// TIA Portal V21 export
FUNCTION "HPHV" : Void   // FC11, LAD
{ S7_Optimized_Access := 'TRUE' }
// stored: SetENOAutomatically false
   VAR_TEMP
      "HOLD START" : Bool;
   END_VAR
   VAR_TEMP   // added for the SCL form of the ladder/FBD networks
      _w1 : Bool;
      _w2 : Bool;
      _w3 : Bool;
      _w4 : Bool;
   END_VAR
BEGIN

REGION Network 1
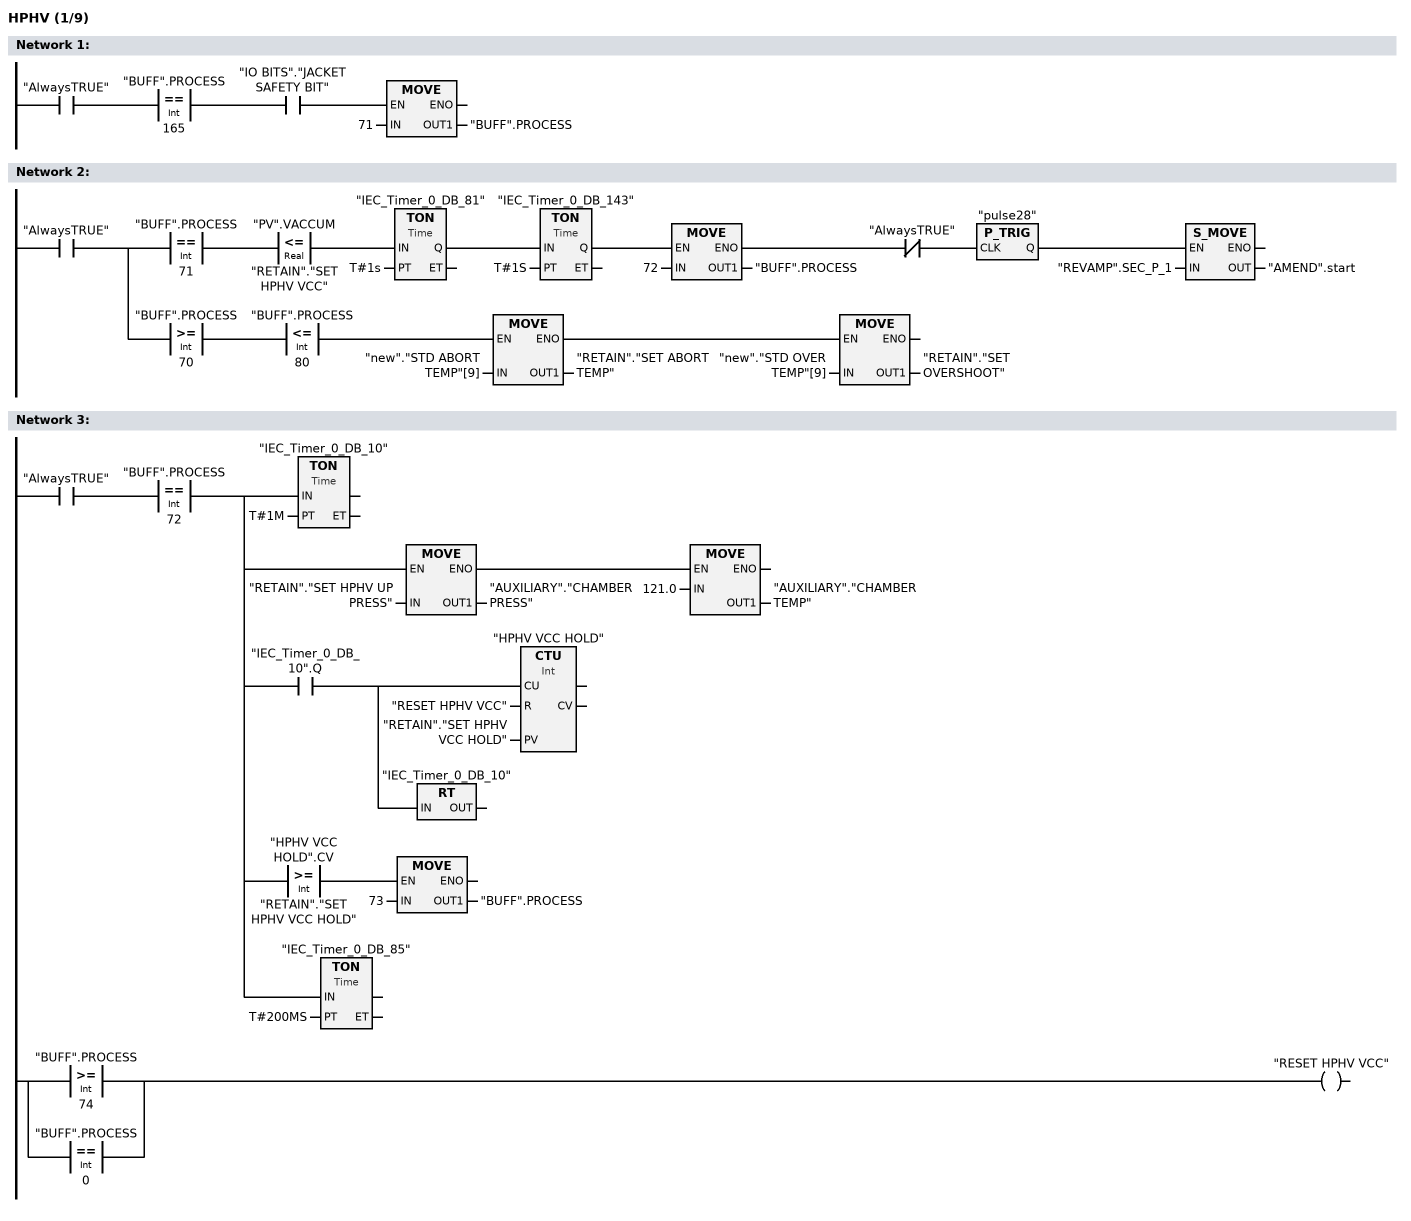
   RUNG wire#powerrail
      Contact( "AlwaysTRUE" )
      { S7_Templates := "SrcType := Int" } EQ_Contact(in1 := "BUFF".PROCESS, in2 := 165)
      Contact( "IO BITS"."JACKET SAFETY BIT" )
      Move(in := 71, out1 => "BUFF".PROCESS)
   END_RUNG
   // the same network as SCL:
   IF "AlwaysTRUE" AND ("BUFF".PROCESS = 165) AND "IO BITS"."JACKET SAFETY BIT" THEN
       "BUFF".PROCESS := 71;
   END_IF;
END_REGION

REGION Network 2
   RUNG wire#powerrail
      Contact( "AlwaysTRUE" )
      wire#w1
      { S7_Templates := "SrcType := Int" } EQ_Contact(in1 := "BUFF".PROCESS, in2 := 71)
      { S7_Templates := "SrcType := Real" } LE_Contact(in1 := "PV".VACCUM, in2 := "RETAIN"."SET HPHV VCC")
      { S7_Templates := "time_type := Time" } "IEC_Timer_0_DB_81".TON(pt := T#1s, et =>)
      { S7_Templates := "time_type := Time" } "IEC_Timer_0_DB_143".TON(pt := T#1S, et =>)
      Move(in := 72, out1 => "BUFF".PROCESS)
      I_Contact( "AlwaysTRUE" )
      P_Trig( "pulse28" )
      S_Move(in := "REVAMP".SEC_P_1, out => "AMEND".start)
   END_RUNG
   RUNG wire#w1
      { S7_Templates := "SrcType := Int" } GE_Contact(in1 := "BUFF".PROCESS, in2 := 70)
      { S7_Templates := "SrcType := Int" } LE_Contact(in1 := "BUFF".PROCESS, in2 := 80)
      Move(in := "new"."STD ABORT TEMP"[9], out1 => "RETAIN"."SET ABORT TEMP")
      Move(in := "new"."STD OVER TEMP"[9], out1 => "RETAIN"."SET OVERSHOOT")
   END_RUNG
   // the same network as SCL:
   "IEC_Timer_0_DB_81".TON(IN := "AlwaysTRUE" AND ("BUFF".PROCESS = 71) AND ("PV".VACCUM <= "RETAIN"."SET HPHV VCC"),
                           PT := T#1s);
   "IEC_Timer_0_DB_143".TON(IN := "IEC_Timer_0_DB_81".Q, PT := T#1S);
   IF "IEC_Timer_0_DB_143".Q THEN "BUFF".PROCESS := 72; END_IF;
   #_w1 := "IEC_Timer_0_DB_143".Q AND NOT "AlwaysTRUE";
   #_w2 := #_w1 AND NOT "pulse28";   // rising edge
   "pulse28" := #_w1;
   IF #_w2 THEN "AMEND".start := "REVAMP".SEC_P_1; END_IF;
   IF "AlwaysTRUE" AND ("BUFF".PROCESS >= 70) AND ("BUFF".PROCESS <= 80) THEN
       "RETAIN"."SET ABORT TEMP" := "new"."STD ABORT TEMP"[9];
       "RETAIN"."SET OVERSHOOT" := "new"."STD OVER TEMP"[9];
   END_IF;
END_REGION

REGION Network 3
   RUNG wire#powerrail
      Contact( "AlwaysTRUE" )
      { S7_Templates := "SrcType := Int" } EQ_Contact(in1 := "BUFF".PROCESS, in2 := 72)
      wire#w1
      { S7_Templates := "time_type := Time" } "IEC_Timer_0_DB_10".TON(pt := T#1M, et =>)
   END_RUNG
   RUNG wire#w1
      Move(in := "RETAIN"."SET HPHV UP PRESS", out1 => "AUXILIARY"."CHAMBER PRESS")
      Move(in := 121.0, out1 => "AUXILIARY"."CHAMBER TEMP")
   END_RUNG
   RUNG wire#w1
      Contact( "IEC_Timer_0_DB_10".Q )
      wire#w2
      { S7_Templates := "value_type := Int" } "HPHV VCC HOLD".CTU(r := "RESET HPHV VCC", pv := "RETAIN"."SET HPHV VCC HOLD", cv =>)
   END_RUNG
   RUNG wire#w2
      RT_Coil( "IEC_Timer_0_DB_10" )
   END_RUNG
   RUNG wire#w1
      { S7_Templates := "SrcType := Int" } GE_Contact(in1 := "HPHV VCC HOLD".CV, in2 := "RETAIN"."SET HPHV VCC HOLD")
      Move(in := 73, out1 => "BUFF".PROCESS)
   END_RUNG
   RUNG wire#w1
      { S7_Templates := "time_type := Time" } "IEC_Timer_0_DB_85".TON(pt := T#200MS, et =>)
   END_RUNG
   RUNG wire#powerrail
      { S7_Templates := "SrcType := Int" } GE_Contact(in1 := "BUFF".PROCESS, in2 := 74)
      wire#w3
      Coil( "RESET HPHV VCC" )
   END_RUNG
   RUNG wire#powerrail
      { S7_Templates := "SrcType := Int" } EQ_Contact(in1 := "BUFF".PROCESS, in2 := 0)
   END_RUNG wire#w3
   // the same network as SCL:
   #_w1 := "AlwaysTRUE" AND ("BUFF".PROCESS = 72);
   "IEC_Timer_0_DB_10".TON(IN := #_w1, PT := T#1M);
   IF #_w1 THEN
       "AUXILIARY"."CHAMBER PRESS" := "RETAIN"."SET HPHV UP PRESS";
       "AUXILIARY"."CHAMBER TEMP" := 121.0;
   END_IF;
   #_w2 := #_w1 AND "IEC_Timer_0_DB_10".Q;
   "HPHV VCC HOLD".CTU(CU := #_w2, R := "RESET HPHV VCC", PV := "RETAIN"."SET HPHV VCC HOLD");
   IF #_w2 THEN RESET_TIMER("IEC_Timer_0_DB_10"); END_IF;
   IF #_w1 AND ("HPHV VCC HOLD".CV >= "RETAIN"."SET HPHV VCC HOLD") THEN "BUFF".PROCESS := 73; END_IF;
   "IEC_Timer_0_DB_85".TON(IN := #_w1, PT := T#200MS);
   "RESET HPHV VCC" := ("BUFF".PROCESS >= 74) OR ("BUFF".PROCESS = 0);
END_REGION

REGION Network 4
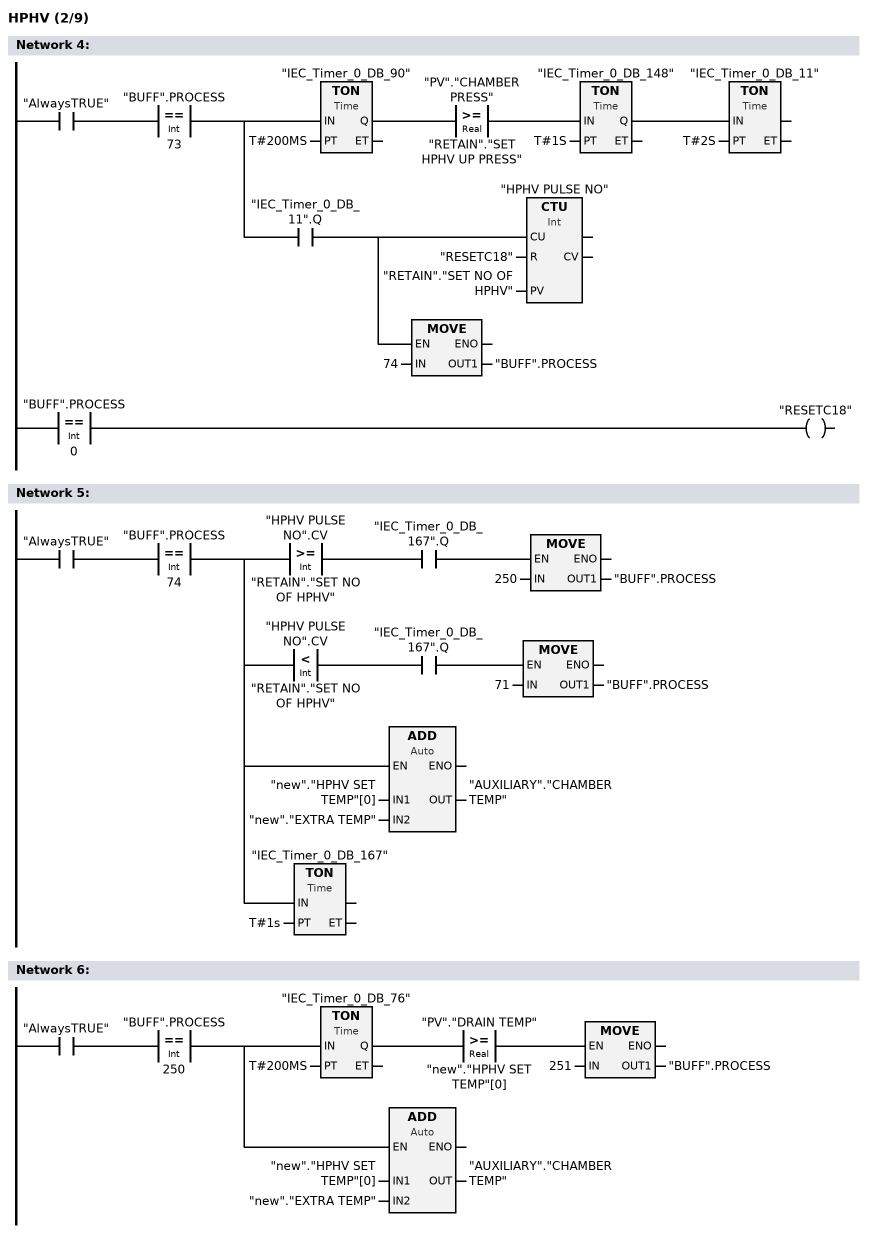
   RUNG wire#powerrail
      Contact( "AlwaysTRUE" )
      { S7_Templates := "SrcType := Int" } EQ_Contact(in1 := "BUFF".PROCESS, in2 := 73)
      wire#w1
      { S7_Templates := "time_type := Time" } "IEC_Timer_0_DB_90".TON(pt := T#200MS, et =>)
      { S7_Templates := "SrcType := Real" } GE_Contact(in1 := "PV"."CHAMBER PRESS", in2 := "RETAIN"."SET HPHV UP PRESS")
      { S7_Templates := "time_type := Time" } "IEC_Timer_0_DB_148".TON(pt := T#1S, et =>)
      { S7_Templates := "time_type := Time" } "IEC_Timer_0_DB_11".TON(pt := T#2S, et =>)
   END_RUNG
   RUNG wire#w1
      Contact( "IEC_Timer_0_DB_11".Q )
      wire#w2
      { S7_Templates := "value_type := Int" } "HPHV PULSE NO".CTU(r := "RESETC18", pv := "RETAIN"."SET NO OF HPHV", cv =>)
   END_RUNG
   RUNG wire#w2
      Move(in := 74, out1 => "BUFF".PROCESS)
   END_RUNG
   RUNG wire#powerrail
      { S7_Templates := "SrcType := Int" } EQ_Contact(in1 := "BUFF".PROCESS, in2 := 0)
      Coil( "RESETC18" )
   END_RUNG
   // the same network as SCL:
   #_w1 := "AlwaysTRUE" AND ("BUFF".PROCESS = 73);
   "IEC_Timer_0_DB_90".TON(IN := #_w1, PT := T#200MS);
   "IEC_Timer_0_DB_148".TON(IN := "IEC_Timer_0_DB_90".Q AND ("PV"."CHAMBER PRESS" >= "RETAIN"."SET HPHV UP PRESS"),
                           PT := T#1S);
   "IEC_Timer_0_DB_11".TON(IN := "IEC_Timer_0_DB_148".Q, PT := T#2S);
   #_w2 := #_w1 AND "IEC_Timer_0_DB_11".Q;
   "HPHV PULSE NO".CTU(CU := #_w2, R := "RESETC18", PV := "RETAIN"."SET NO OF HPHV");
   IF #_w2 THEN "BUFF".PROCESS := 74; END_IF;
   "RESETC18" := "BUFF".PROCESS = 0;
END_REGION

REGION Network 5
   RUNG wire#powerrail
      Contact( "AlwaysTRUE" )
      { S7_Templates := "SrcType := Int" } EQ_Contact(in1 := "BUFF".PROCESS, in2 := 74)
      wire#w1
      { S7_Templates := "SrcType := Int" } GE_Contact(in1 := "HPHV PULSE NO".CV, in2 := "RETAIN"."SET NO OF HPHV")
      Contact( "IEC_Timer_0_DB_167".Q )
      Move(in := 250, out1 => "BUFF".PROCESS)
   END_RUNG
   RUNG wire#w1
      { S7_Templates := "SrcType := Int" } LT_Contact(in1 := "HPHV PULSE NO".CV, in2 := "RETAIN"."SET NO OF HPHV")
      Contact( "IEC_Timer_0_DB_167".Q )
      Move(in := 71, out1 => "BUFF".PROCESS)
   END_RUNG
   RUNG wire#w1
      Add(in1 := "new"."HPHV SET TEMP"[0], in2 := "new"."EXTRA TEMP", out => "AUXILIARY"."CHAMBER TEMP")
   END_RUNG
   RUNG wire#w1
      { S7_Templates := "time_type := Time" } "IEC_Timer_0_DB_167".TON(pt := T#1s, et =>)
   END_RUNG
   // the same network as SCL:
   #_w1 := "AlwaysTRUE" AND ("BUFF".PROCESS = 74);
   IF #_w1 AND ("HPHV PULSE NO".CV >= "RETAIN"."SET NO OF HPHV") AND "IEC_Timer_0_DB_167".Q THEN
       "BUFF".PROCESS := 250;
   END_IF;
   IF #_w1 AND ("HPHV PULSE NO".CV < "RETAIN"."SET NO OF HPHV") AND "IEC_Timer_0_DB_167".Q THEN
       "BUFF".PROCESS := 71;
   END_IF;
   IF #_w1 THEN "AUXILIARY"."CHAMBER TEMP" := "new"."HPHV SET TEMP"[0] + "new"."EXTRA TEMP"; END_IF;
   "IEC_Timer_0_DB_167".TON(IN := #_w1, PT := T#1s);
END_REGION

REGION Network 6
   RUNG wire#powerrail
      Contact( "AlwaysTRUE" )
      { S7_Templates := "SrcType := Int" } EQ_Contact(in1 := "BUFF".PROCESS, in2 := 250)
      wire#w1
      { S7_Templates := "time_type := Time" } "IEC_Timer_0_DB_76".TON(pt := T#200MS, et =>)
      { S7_Templates := "SrcType := Real" } GE_Contact(in1 := "PV"."DRAIN TEMP", in2 := "new"."HPHV SET TEMP"[0])
      Move(in := 251, out1 => "BUFF".PROCESS)
   END_RUNG
   RUNG wire#w1
      Add(in1 := "new"."HPHV SET TEMP"[0], in2 := "new"."EXTRA TEMP", out => "AUXILIARY"."CHAMBER TEMP")
   END_RUNG
   // the same network as SCL:
   #_w1 := "AlwaysTRUE" AND ("BUFF".PROCESS = 250);
   "IEC_Timer_0_DB_76".TON(IN := #_w1, PT := T#200MS);
   IF "IEC_Timer_0_DB_76".Q AND ("PV"."DRAIN TEMP" >= "new"."HPHV SET TEMP"[0]) THEN
       "BUFF".PROCESS := 251;
   END_IF;
   IF #_w1 THEN "AUXILIARY"."CHAMBER TEMP" := "new"."HPHV SET TEMP"[0] + "new"."EXTRA TEMP"; END_IF;
END_REGION

REGION Network 7
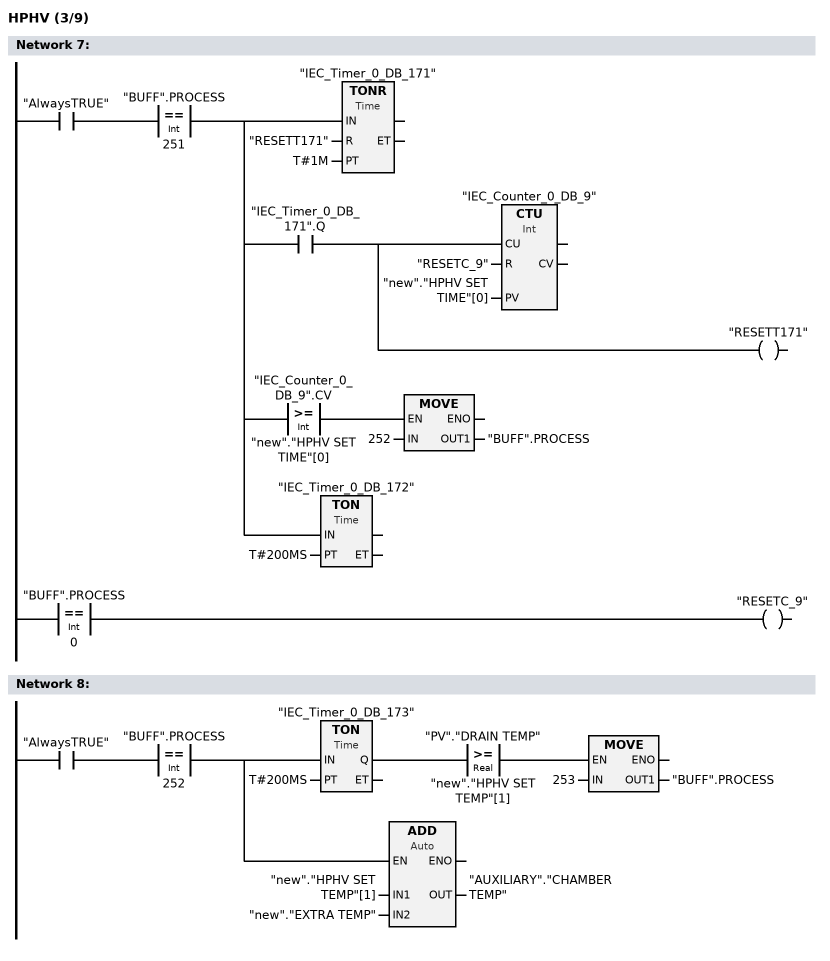
   RUNG wire#powerrail
      Contact( "AlwaysTRUE" )
      { S7_Templates := "SrcType := Int" } EQ_Contact(in1 := "BUFF".PROCESS, in2 := 251)
      wire#w1
      { S7_Templates := "time_type := Time" } "IEC_Timer_0_DB_171".TONR(r := "RESETT171", pt := T#1M, et =>)
   END_RUNG
   RUNG wire#w1
      Contact( "IEC_Timer_0_DB_171".Q )
      wire#w2
      { S7_Templates := "value_type := Int" } "IEC_Counter_0_DB_9".CTU(r := "RESETC_9", pv := "new"."HPHV SET TIME"[0], cv =>)
   END_RUNG
   RUNG wire#w2
      Coil( "RESETT171" )
   END_RUNG
   RUNG wire#w1
      { S7_Templates := "SrcType := Int" } GE_Contact(in1 := "IEC_Counter_0_DB_9".CV, in2 := "new"."HPHV SET TIME"[0])
      Move(in := 252, out1 => "BUFF".PROCESS)
   END_RUNG
   RUNG wire#w1
      { S7_Templates := "time_type := Time" } "IEC_Timer_0_DB_172".TON(pt := T#200MS, et =>)
   END_RUNG
   RUNG wire#powerrail
      { S7_Templates := "SrcType := Int" } EQ_Contact(in1 := "BUFF".PROCESS, in2 := 0)
      Coil( "RESETC_9" )
   END_RUNG
   // the same network as SCL:
   #_w1 := "AlwaysTRUE" AND ("BUFF".PROCESS = 251);
   "IEC_Timer_0_DB_171".TONR(IN := #_w1, R := "RESETT171", PT := T#1M);
   #_w2 := #_w1 AND "IEC_Timer_0_DB_171".Q;
   "IEC_Counter_0_DB_9".CTU(CU := #_w2, R := "RESETC_9", PV := "new"."HPHV SET TIME"[0]);
   "RESETT171" := #_w2;
   IF #_w1 AND ("IEC_Counter_0_DB_9".CV >= "new"."HPHV SET TIME"[0]) THEN "BUFF".PROCESS := 252; END_IF;
   "IEC_Timer_0_DB_172".TON(IN := #_w1, PT := T#200MS);
   "RESETC_9" := "BUFF".PROCESS = 0;
END_REGION

REGION Network 8
   RUNG wire#powerrail
      Contact( "AlwaysTRUE" )
      { S7_Templates := "SrcType := Int" } EQ_Contact(in1 := "BUFF".PROCESS, in2 := 252)
      wire#w1
      { S7_Templates := "time_type := Time" } "IEC_Timer_0_DB_173".TON(pt := T#200MS, et =>)
      { S7_Templates := "SrcType := Real" } GE_Contact(in1 := "PV"."DRAIN TEMP", in2 := "new"."HPHV SET TEMP"[1])
      Move(in := 253, out1 => "BUFF".PROCESS)
   END_RUNG
   RUNG wire#w1
      Add(in1 := "new"."HPHV SET TEMP"[1], in2 := "new"."EXTRA TEMP", out => "AUXILIARY"."CHAMBER TEMP")
   END_RUNG
   // the same network as SCL:
   #_w1 := "AlwaysTRUE" AND ("BUFF".PROCESS = 252);
   "IEC_Timer_0_DB_173".TON(IN := #_w1, PT := T#200MS);
   IF "IEC_Timer_0_DB_173".Q AND ("PV"."DRAIN TEMP" >= "new"."HPHV SET TEMP"[1]) THEN
       "BUFF".PROCESS := 253;
   END_IF;
   IF #_w1 THEN "AUXILIARY"."CHAMBER TEMP" := "new"."HPHV SET TEMP"[1] + "new"."EXTRA TEMP"; END_IF;
END_REGION

REGION Network 9
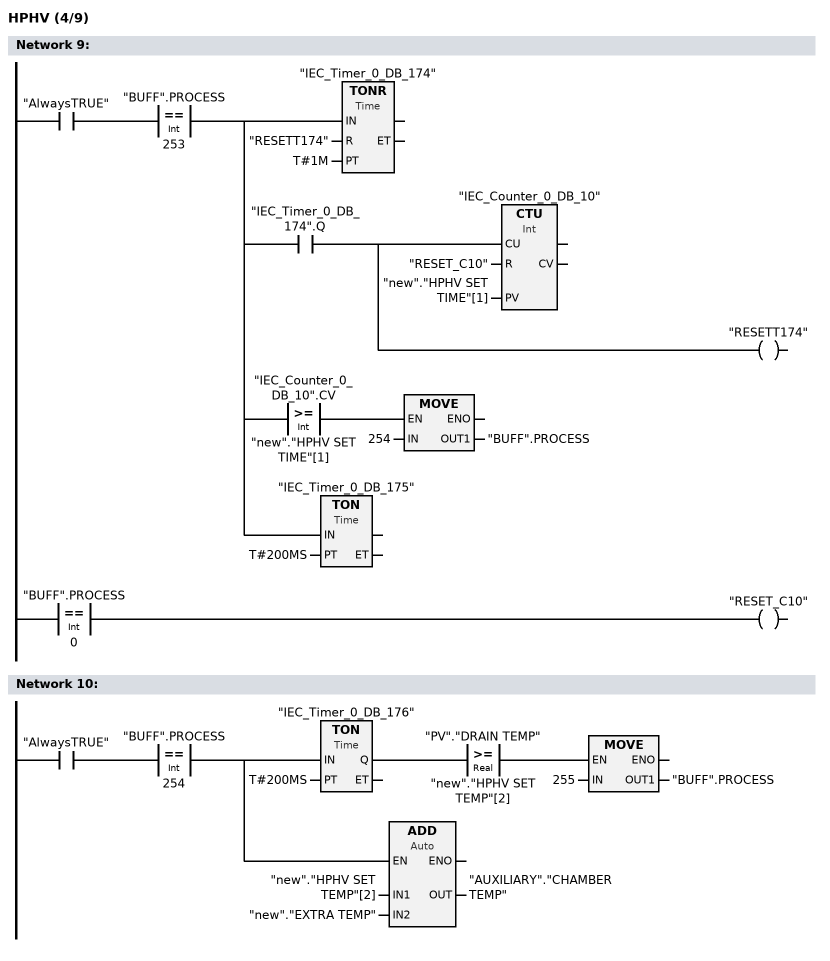
   RUNG wire#powerrail
      Contact( "AlwaysTRUE" )
      { S7_Templates := "SrcType := Int" } EQ_Contact(in1 := "BUFF".PROCESS, in2 := 253)
      wire#w1
      { S7_Templates := "time_type := Time" } "IEC_Timer_0_DB_174".TONR(r := "RESETT174", pt := T#1M, et =>)
   END_RUNG
   RUNG wire#w1
      Contact( "IEC_Timer_0_DB_174".Q )
      wire#w2
      { S7_Templates := "value_type := Int" } "IEC_Counter_0_DB_10".CTU(r := "RESET_C10", pv := "new"."HPHV SET TIME"[1], cv =>)
   END_RUNG
   RUNG wire#w2
      Coil( "RESETT174" )
   END_RUNG
   RUNG wire#w1
      { S7_Templates := "SrcType := Int" } GE_Contact(in1 := "IEC_Counter_0_DB_10".CV, in2 := "new"."HPHV SET TIME"[1])
      Move(in := 254, out1 => "BUFF".PROCESS)
   END_RUNG
   RUNG wire#w1
      { S7_Templates := "time_type := Time" } "IEC_Timer_0_DB_175".TON(pt := T#200MS, et =>)
   END_RUNG
   RUNG wire#powerrail
      { S7_Templates := "SrcType := Int" } EQ_Contact(in1 := "BUFF".PROCESS, in2 := 0)
      Coil( "RESET_C10" )
   END_RUNG
   // the same network as SCL:
   #_w1 := "AlwaysTRUE" AND ("BUFF".PROCESS = 253);
   "IEC_Timer_0_DB_174".TONR(IN := #_w1, R := "RESETT174", PT := T#1M);
   #_w2 := #_w1 AND "IEC_Timer_0_DB_174".Q;
   "IEC_Counter_0_DB_10".CTU(CU := #_w2, R := "RESET_C10", PV := "new"."HPHV SET TIME"[1]);
   "RESETT174" := #_w2;
   IF #_w1 AND ("IEC_Counter_0_DB_10".CV >= "new"."HPHV SET TIME"[1]) THEN "BUFF".PROCESS := 254; END_IF;
   "IEC_Timer_0_DB_175".TON(IN := #_w1, PT := T#200MS);
   "RESET_C10" := "BUFF".PROCESS = 0;
END_REGION

REGION Network 10
   RUNG wire#powerrail
      Contact( "AlwaysTRUE" )
      { S7_Templates := "SrcType := Int" } EQ_Contact(in1 := "BUFF".PROCESS, in2 := 254)
      wire#w1
      { S7_Templates := "time_type := Time" } "IEC_Timer_0_DB_176".TON(pt := T#200MS, et =>)
      { S7_Templates := "SrcType := Real" } GE_Contact(in1 := "PV"."DRAIN TEMP", in2 := "new"."HPHV SET TEMP"[2])
      Move(in := 255, out1 => "BUFF".PROCESS)
   END_RUNG
   RUNG wire#w1
      Add(in1 := "new"."HPHV SET TEMP"[2], in2 := "new"."EXTRA TEMP", out => "AUXILIARY"."CHAMBER TEMP")
   END_RUNG
   // the same network as SCL:
   #_w1 := "AlwaysTRUE" AND ("BUFF".PROCESS = 254);
   "IEC_Timer_0_DB_176".TON(IN := #_w1, PT := T#200MS);
   IF "IEC_Timer_0_DB_176".Q AND ("PV"."DRAIN TEMP" >= "new"."HPHV SET TEMP"[2]) THEN
       "BUFF".PROCESS := 255;
   END_IF;
   IF #_w1 THEN "AUXILIARY"."CHAMBER TEMP" := "new"."HPHV SET TEMP"[2] + "new"."EXTRA TEMP"; END_IF;
END_REGION

REGION Network 11
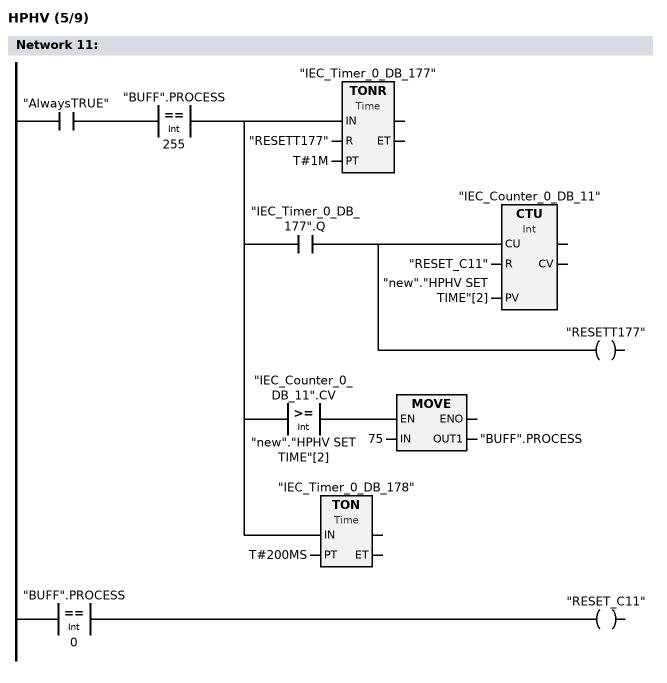
   RUNG wire#powerrail
      Contact( "AlwaysTRUE" )
      { S7_Templates := "SrcType := Int" } EQ_Contact(in1 := "BUFF".PROCESS, in2 := 255)
      wire#w1
      { S7_Templates := "time_type := Time" } "IEC_Timer_0_DB_177".TONR(r := "RESETT177", pt := T#1M, et =>)
   END_RUNG
   RUNG wire#w1
      Contact( "IEC_Timer_0_DB_177".Q )
      wire#w2
      { S7_Templates := "value_type := Int" } "IEC_Counter_0_DB_11".CTU(r := "RESET_C11", pv := "new"."HPHV SET TIME"[2], cv =>)
   END_RUNG
   RUNG wire#w2
      Coil( "RESETT177" )
   END_RUNG
   RUNG wire#w1
      { S7_Templates := "SrcType := Int" } GE_Contact(in1 := "IEC_Counter_0_DB_11".CV, in2 := "new"."HPHV SET TIME"[2])
      Move(in := 75, out1 => "BUFF".PROCESS)
   END_RUNG
   RUNG wire#w1
      { S7_Templates := "time_type := Time" } "IEC_Timer_0_DB_178".TON(pt := T#200MS, et =>)
   END_RUNG
   RUNG wire#powerrail
      { S7_Templates := "SrcType := Int" } EQ_Contact(in1 := "BUFF".PROCESS, in2 := 0)
      Coil( "RESET_C11" )
   END_RUNG
   // the same network as SCL:
   #_w1 := "AlwaysTRUE" AND ("BUFF".PROCESS = 255);
   "IEC_Timer_0_DB_177".TONR(IN := #_w1, R := "RESETT177", PT := T#1M);
   #_w2 := #_w1 AND "IEC_Timer_0_DB_177".Q;
   "IEC_Counter_0_DB_11".CTU(CU := #_w2, R := "RESET_C11", PV := "new"."HPHV SET TIME"[2]);
   "RESETT177" := #_w2;
   IF #_w1 AND ("IEC_Counter_0_DB_11".CV >= "new"."HPHV SET TIME"[2]) THEN "BUFF".PROCESS := 75; END_IF;
   "IEC_Timer_0_DB_178".TON(IN := #_w1, PT := T#200MS);
   "RESET_C11" := "BUFF".PROCESS = 0;
END_REGION

REGION Network 12
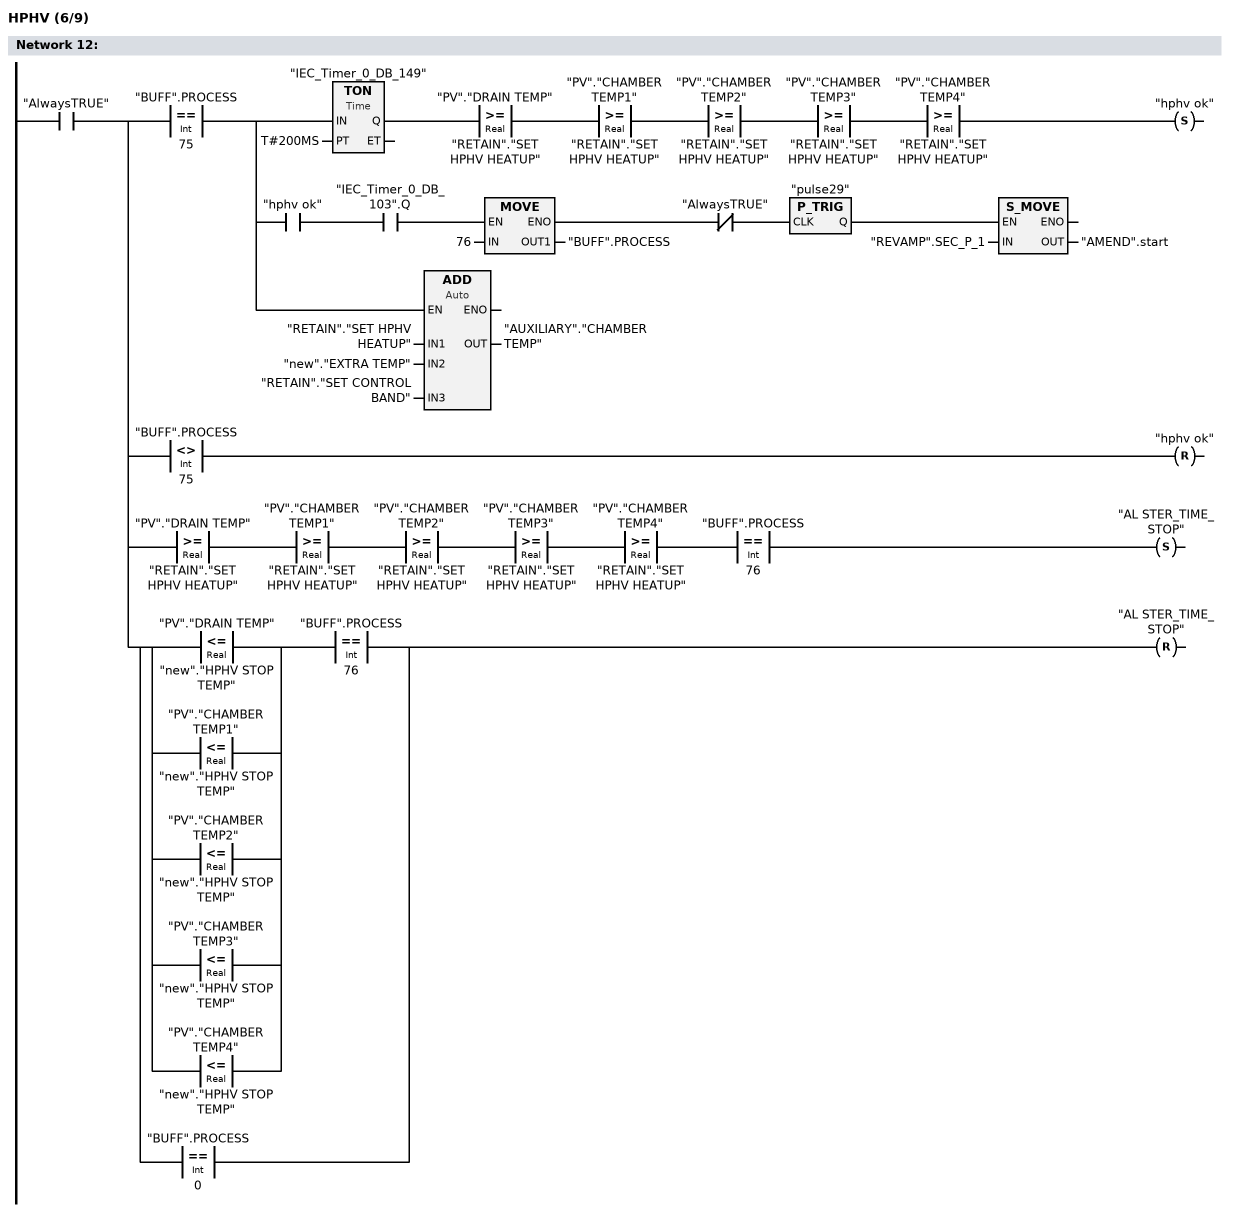
   RUNG wire#powerrail
      Contact( "AlwaysTRUE" )
      wire#w1
      { S7_Templates := "SrcType := Int" } EQ_Contact(in1 := "BUFF".PROCESS, in2 := 75)
      wire#w2
      { S7_Templates := "time_type := Time" } "IEC_Timer_0_DB_149".TON(pt := T#200MS, et =>)
      { S7_Templates := "SrcType := Real" } GE_Contact(in1 := "PV"."DRAIN TEMP", in2 := "RETAIN"."SET HPHV HEATUP")
      { S7_Templates := "SrcType := Real" } GE_Contact(in1 := "PV"."CHAMBER TEMP1", in2 := "RETAIN"."SET HPHV HEATUP")
      { S7_Templates := "SrcType := Real" } GE_Contact(in1 := "PV"."CHAMBER TEMP2", in2 := "RETAIN"."SET HPHV HEATUP")
      { S7_Templates := "SrcType := Real" } GE_Contact(in1 := "PV"."CHAMBER TEMP3", in2 := "RETAIN"."SET HPHV HEATUP")
      { S7_Templates := "SrcType := Real" } GE_Contact(in1 := "PV"."CHAMBER TEMP4", in2 := "RETAIN"."SET HPHV HEATUP")
      S_Coil( "hphv ok" )
   END_RUNG
   RUNG wire#w2
      Contact( "hphv ok" )
      Contact( "IEC_Timer_0_DB_103".Q )
      Move(in := 76, out1 => "BUFF".PROCESS)
      I_Contact( "AlwaysTRUE" )
      P_Trig( "pulse29" )
      S_Move(in := "REVAMP".SEC_P_1, out => "AMEND".start)
   END_RUNG
   RUNG wire#w2
      Add(in1 := "RETAIN"."SET HPHV HEATUP", in2 := "new"."EXTRA TEMP", in3 := "RETAIN"."SET CONTROL BAND", out => "AUXILIARY"."CHAMBER TEMP")
   END_RUNG
   RUNG wire#w1
      { S7_Templates := "SrcType := Int" } NE_Contact(in1 := "BUFF".PROCESS, in2 := 75)
      R_Coil( "hphv ok" )
   END_RUNG
   RUNG wire#w1
      { S7_Templates := "SrcType := Real" } GE_Contact(in1 := "PV"."DRAIN TEMP", in2 := "RETAIN"."SET HPHV HEATUP")
      { S7_Templates := "SrcType := Real" } GE_Contact(in1 := "PV"."CHAMBER TEMP1", in2 := "RETAIN"."SET HPHV HEATUP")
      { S7_Templates := "SrcType := Real" } GE_Contact(in1 := "PV"."CHAMBER TEMP2", in2 := "RETAIN"."SET HPHV HEATUP")
      { S7_Templates := "SrcType := Real" } GE_Contact(in1 := "PV"."CHAMBER TEMP3", in2 := "RETAIN"."SET HPHV HEATUP")
      { S7_Templates := "SrcType := Real" } GE_Contact(in1 := "PV"."CHAMBER TEMP4", in2 := "RETAIN"."SET HPHV HEATUP")
      { S7_Templates := "SrcType := Int" } EQ_Contact(in1 := "BUFF".PROCESS, in2 := 76)
      S_Coil( "AL STER_TIME_STOP" )
   END_RUNG
   RUNG wire#w1
      { S7_Templates := "SrcType := Real" } LE_Contact(in1 := "PV"."DRAIN TEMP", in2 := "new"."HPHV STOP TEMP")
      wire#w3
      { S7_Templates := "SrcType := Int" } EQ_Contact(in1 := "BUFF".PROCESS, in2 := 76)
      wire#w4
      R_Coil( "AL STER_TIME_STOP" )
   END_RUNG
   RUNG wire#w1
      { S7_Templates := "SrcType := Real" } LE_Contact(in1 := "PV"."CHAMBER TEMP1", in2 := "new"."HPHV STOP TEMP")
   END_RUNG wire#w3
   RUNG wire#w1
      { S7_Templates := "SrcType := Real" } LE_Contact(in1 := "PV"."CHAMBER TEMP2", in2 := "new"."HPHV STOP TEMP")
   END_RUNG wire#w3
   RUNG wire#w1
      { S7_Templates := "SrcType := Real" } LE_Contact(in1 := "PV"."CHAMBER TEMP3", in2 := "new"."HPHV STOP TEMP")
   END_RUNG wire#w3
   RUNG wire#w1
      { S7_Templates := "SrcType := Real" } LE_Contact(in1 := "PV"."CHAMBER TEMP4", in2 := "new"."HPHV STOP TEMP")
   END_RUNG wire#w3
   RUNG wire#w1
      { S7_Templates := "SrcType := Int" } EQ_Contact(in1 := "BUFF".PROCESS, in2 := 0)
   END_RUNG wire#w4
   // the same network as SCL:
   #_w1 := "AlwaysTRUE" AND ("BUFF".PROCESS = 75);
   "IEC_Timer_0_DB_149".TON(IN := #_w1, PT := T#200MS);
   IF "IEC_Timer_0_DB_149".Q AND ("PV"."DRAIN TEMP" >= "RETAIN"."SET HPHV HEATUP") AND ("PV"."CHAMBER TEMP1" >= "RETAIN"."SET HPHV HEATUP") AND ("PV"."CHAMBER TEMP2" >= "RETAIN"."SET HPHV HEATUP") AND ("PV"."CHAMBER TEMP3" >= "RETAIN"."SET HPHV HEATUP") AND ("PV"."CHAMBER TEMP4" >= "RETAIN"."SET HPHV HEATUP") THEN
       "hphv ok" := TRUE;
   END_IF;
   #_w2 := #_w1 AND "hphv ok" AND "IEC_Timer_0_DB_103".Q;
   IF #_w2 THEN "BUFF".PROCESS := 76; END_IF;
   #_w3 := #_w2 AND NOT "AlwaysTRUE";
   #_w4 := #_w3 AND NOT "pulse29";   // rising edge
   "pulse29" := #_w3;
   IF #_w4 THEN "AMEND".start := "REVAMP".SEC_P_1; END_IF;
   IF #_w1 THEN
       "AUXILIARY"."CHAMBER TEMP" := "RETAIN"."SET HPHV HEATUP" + "new"."EXTRA TEMP" + "RETAIN"."SET CONTROL BAND";
   END_IF;
   IF "AlwaysTRUE" AND ("BUFF".PROCESS <> 75) THEN "hphv ok" := FALSE; END_IF;
   IF "AlwaysTRUE" AND ("PV"."DRAIN TEMP" >= "RETAIN"."SET HPHV HEATUP") AND ("PV"."CHAMBER TEMP1" >= "RETAIN"."SET HPHV HEATUP") AND ("PV"."CHAMBER TEMP2" >= "RETAIN"."SET HPHV HEATUP") AND ("PV"."CHAMBER TEMP3" >= "RETAIN"."SET HPHV HEATUP") AND ("PV"."CHAMBER TEMP4" >= "RETAIN"."SET HPHV HEATUP") AND ("BUFF".PROCESS = 76) THEN
       "AL STER_TIME_STOP" := TRUE;
   END_IF;
   IF "AlwaysTRUE" AND (((("PV"."DRAIN TEMP" <= "new"."HPHV STOP TEMP") OR ("PV"."CHAMBER TEMP1" <= "new"."HPHV STOP TEMP") OR ("PV"."CHAMBER TEMP2" <= "new"."HPHV STOP TEMP") OR ("PV"."CHAMBER TEMP3" <= "new"."HPHV STOP TEMP") OR ("PV"."CHAMBER TEMP4" <= "new"."HPHV STOP TEMP")) AND ("BUFF".PROCESS = 76)) OR ("BUFF".PROCESS = 0)) THEN
       "AL STER_TIME_STOP" := FALSE;
   END_IF;
END_REGION

REGION Network 13
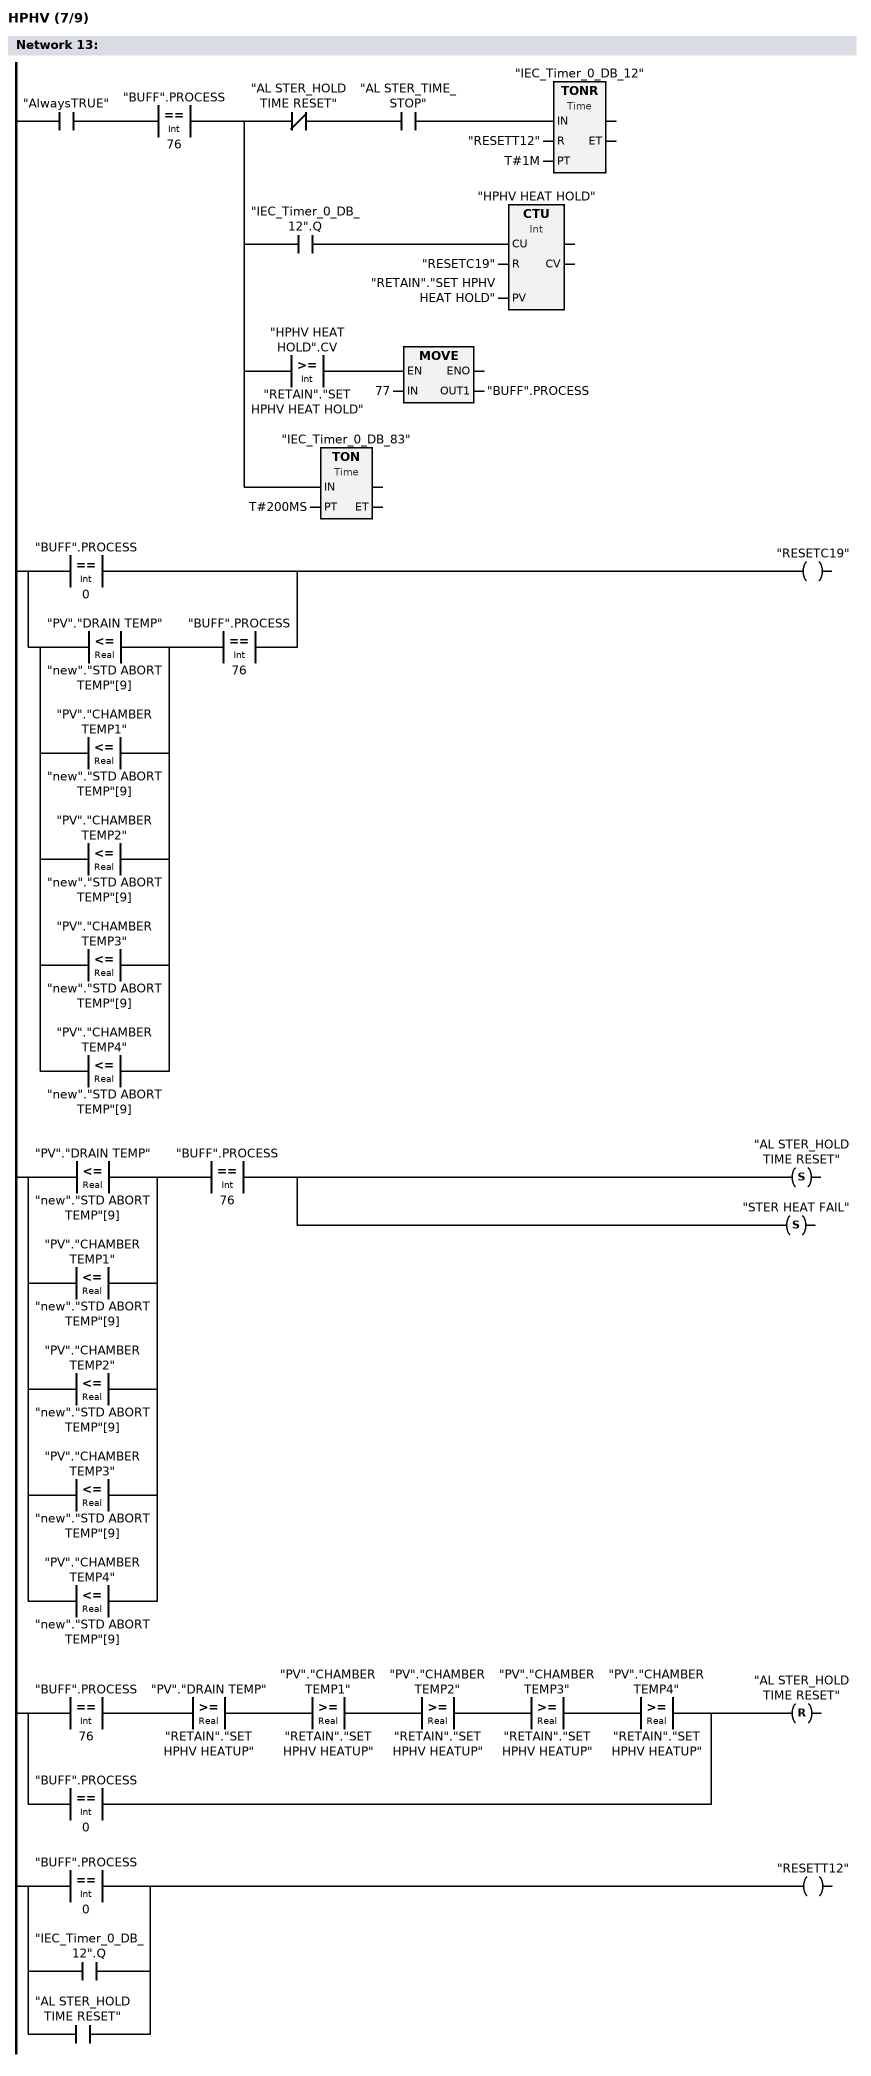
   RUNG wire#powerrail
      Contact( "AlwaysTRUE" )
      { S7_Templates := "SrcType := Int" } EQ_Contact(in1 := "BUFF".PROCESS, in2 := 76)
      wire#w1
      I_Contact( "AL STER_HOLD TIME RESET" )
      Contact( "AL STER_TIME_STOP" )
      { S7_Templates := "time_type := Time" } "IEC_Timer_0_DB_12".TONR(r := "RESETT12", pt := T#1M, et =>)
   END_RUNG
   RUNG wire#w1
      Contact( "IEC_Timer_0_DB_12".Q )
      { S7_Templates := "value_type := Int" } "HPHV HEAT HOLD".CTU(r := "RESETC19", pv := "RETAIN"."SET HPHV HEAT HOLD", cv =>)
   END_RUNG
   RUNG wire#w1
      { S7_Templates := "SrcType := Int" } GE_Contact(in1 := "HPHV HEAT HOLD".CV, in2 := "RETAIN"."SET HPHV HEAT HOLD")
      Move(in := 77, out1 => "BUFF".PROCESS)
   END_RUNG
   RUNG wire#w1
      { S7_Templates := "time_type := Time" } "IEC_Timer_0_DB_83".TON(pt := T#200MS, et =>)
   END_RUNG
   RUNG wire#powerrail
      { S7_Templates := "SrcType := Int" } EQ_Contact(in1 := "BUFF".PROCESS, in2 := 0)
      wire#w2
      Coil( "RESETC19" )
   END_RUNG
   RUNG wire#powerrail
      { S7_Templates := "SrcType := Real" } LE_Contact(in1 := "PV"."DRAIN TEMP", in2 := "new"."STD ABORT TEMP"[9])
      wire#w3
      { S7_Templates := "SrcType := Int" } EQ_Contact(in1 := "BUFF".PROCESS, in2 := 76)
   END_RUNG wire#w2
   RUNG wire#powerrail
      { S7_Templates := "SrcType := Real" } LE_Contact(in1 := "PV"."CHAMBER TEMP1", in2 := "new"."STD ABORT TEMP"[9])
   END_RUNG wire#w3
   RUNG wire#powerrail
      { S7_Templates := "SrcType := Real" } LE_Contact(in1 := "PV"."CHAMBER TEMP2", in2 := "new"."STD ABORT TEMP"[9])
   END_RUNG wire#w3
   RUNG wire#powerrail
      { S7_Templates := "SrcType := Real" } LE_Contact(in1 := "PV"."CHAMBER TEMP3", in2 := "new"."STD ABORT TEMP"[9])
   END_RUNG wire#w3
   RUNG wire#powerrail
      { S7_Templates := "SrcType := Real" } LE_Contact(in1 := "PV"."CHAMBER TEMP4", in2 := "new"."STD ABORT TEMP"[9])
   END_RUNG wire#w3
   RUNG wire#powerrail
      { S7_Templates := "SrcType := Real" } LE_Contact(in1 := "PV"."DRAIN TEMP", in2 := "new"."STD ABORT TEMP"[9])
      wire#w4
      { S7_Templates := "SrcType := Int" } EQ_Contact(in1 := "BUFF".PROCESS, in2 := 76)
      wire#w5
      S_Coil( "AL STER_HOLD TIME RESET" )
   END_RUNG
   RUNG wire#powerrail
      { S7_Templates := "SrcType := Real" } LE_Contact(in1 := "PV"."CHAMBER TEMP1", in2 := "new"."STD ABORT TEMP"[9])
   END_RUNG wire#w4
   RUNG wire#powerrail
      { S7_Templates := "SrcType := Real" } LE_Contact(in1 := "PV"."CHAMBER TEMP2", in2 := "new"."STD ABORT TEMP"[9])
   END_RUNG wire#w4
   RUNG wire#powerrail
      { S7_Templates := "SrcType := Real" } LE_Contact(in1 := "PV"."CHAMBER TEMP3", in2 := "new"."STD ABORT TEMP"[9])
   END_RUNG wire#w4
   RUNG wire#powerrail
      { S7_Templates := "SrcType := Real" } LE_Contact(in1 := "PV"."CHAMBER TEMP4", in2 := "new"."STD ABORT TEMP"[9])
   END_RUNG wire#w4
   RUNG wire#w5
      S_Coil( "STER HEAT FAIL" )
   END_RUNG
   RUNG wire#powerrail
      { S7_Templates := "SrcType := Int" } EQ_Contact(in1 := "BUFF".PROCESS, in2 := 76)
      { S7_Templates := "SrcType := Real" } GE_Contact(in1 := "PV"."DRAIN TEMP", in2 := "RETAIN"."SET HPHV HEATUP")
      { S7_Templates := "SrcType := Real" } GE_Contact(in1 := "PV"."CHAMBER TEMP1", in2 := "RETAIN"."SET HPHV HEATUP")
      { S7_Templates := "SrcType := Real" } GE_Contact(in1 := "PV"."CHAMBER TEMP2", in2 := "RETAIN"."SET HPHV HEATUP")
      { S7_Templates := "SrcType := Real" } GE_Contact(in1 := "PV"."CHAMBER TEMP3", in2 := "RETAIN"."SET HPHV HEATUP")
      { S7_Templates := "SrcType := Real" } GE_Contact(in1 := "PV"."CHAMBER TEMP4", in2 := "RETAIN"."SET HPHV HEATUP")
      wire#w6
      R_Coil( "AL STER_HOLD TIME RESET" )
   END_RUNG
   RUNG wire#powerrail
      { S7_Templates := "SrcType := Int" } EQ_Contact(in1 := "BUFF".PROCESS, in2 := 0)
   END_RUNG wire#w6
   RUNG wire#powerrail
      { S7_Templates := "SrcType := Int" } EQ_Contact(in1 := "BUFF".PROCESS, in2 := 0)
      wire#w7
      Coil( "RESETT12" )
   END_RUNG
   RUNG wire#powerrail
      Contact( "IEC_Timer_0_DB_12".Q )
   END_RUNG wire#w7
   RUNG wire#powerrail
      Contact( "AL STER_HOLD TIME RESET" )
   END_RUNG wire#w7
   // the same network as SCL:
   #_w1 := "AlwaysTRUE" AND ("BUFF".PROCESS = 76);
   "IEC_Timer_0_DB_12".TONR(IN := #_w1 AND NOT "AL STER_HOLD TIME RESET" AND "AL STER_TIME_STOP",
                           R := "RESETT12",
                           PT := T#1M);
   "HPHV HEAT HOLD".CTU(CU := #_w1 AND "IEC_Timer_0_DB_12".Q,
                        R := "RESETC19",
                        PV := "RETAIN"."SET HPHV HEAT HOLD");
   IF #_w1 AND ("HPHV HEAT HOLD".CV >= "RETAIN"."SET HPHV HEAT HOLD") THEN "BUFF".PROCESS := 77; END_IF;
   "IEC_Timer_0_DB_83".TON(IN := #_w1, PT := T#200MS);
   "RESETC19" := ("BUFF".PROCESS = 0) OR ((("PV"."DRAIN TEMP" <= "new"."STD ABORT TEMP"[9]) OR ("PV"."CHAMBER TEMP1" <= "new"."STD ABORT TEMP"[9]) OR ("PV"."CHAMBER TEMP2" <= "new"."STD ABORT TEMP"[9]) OR ("PV"."CHAMBER TEMP3" <= "new"."STD ABORT TEMP"[9]) OR ("PV"."CHAMBER TEMP4" <= "new"."STD ABORT TEMP"[9])) AND ("BUFF".PROCESS = 76));
   IF (("PV"."DRAIN TEMP" <= "new"."STD ABORT TEMP"[9]) OR ("PV"."CHAMBER TEMP1" <= "new"."STD ABORT TEMP"[9]) OR ("PV"."CHAMBER TEMP2" <= "new"."STD ABORT TEMP"[9]) OR ("PV"."CHAMBER TEMP3" <= "new"."STD ABORT TEMP"[9]) OR ("PV"."CHAMBER TEMP4" <= "new"."STD ABORT TEMP"[9])) AND ("BUFF".PROCESS = 76) THEN
       "AL STER_HOLD TIME RESET" := TRUE;
       "STER HEAT FAIL" := TRUE;
   END_IF;
   IF (("BUFF".PROCESS = 76) AND ("PV"."DRAIN TEMP" >= "RETAIN"."SET HPHV HEATUP") AND ("PV"."CHAMBER TEMP1" >= "RETAIN"."SET HPHV HEATUP") AND ("PV"."CHAMBER TEMP2" >= "RETAIN"."SET HPHV HEATUP") AND ("PV"."CHAMBER TEMP3" >= "RETAIN"."SET HPHV HEATUP") AND ("PV"."CHAMBER TEMP4" >= "RETAIN"."SET HPHV HEATUP")) OR ("BUFF".PROCESS = 0) THEN
       "AL STER_HOLD TIME RESET" := FALSE;
   END_IF;
   "RESETT12" := ("BUFF".PROCESS = 0) OR "IEC_Timer_0_DB_12".Q OR "AL STER_HOLD TIME RESET";
END_REGION

REGION Network 14
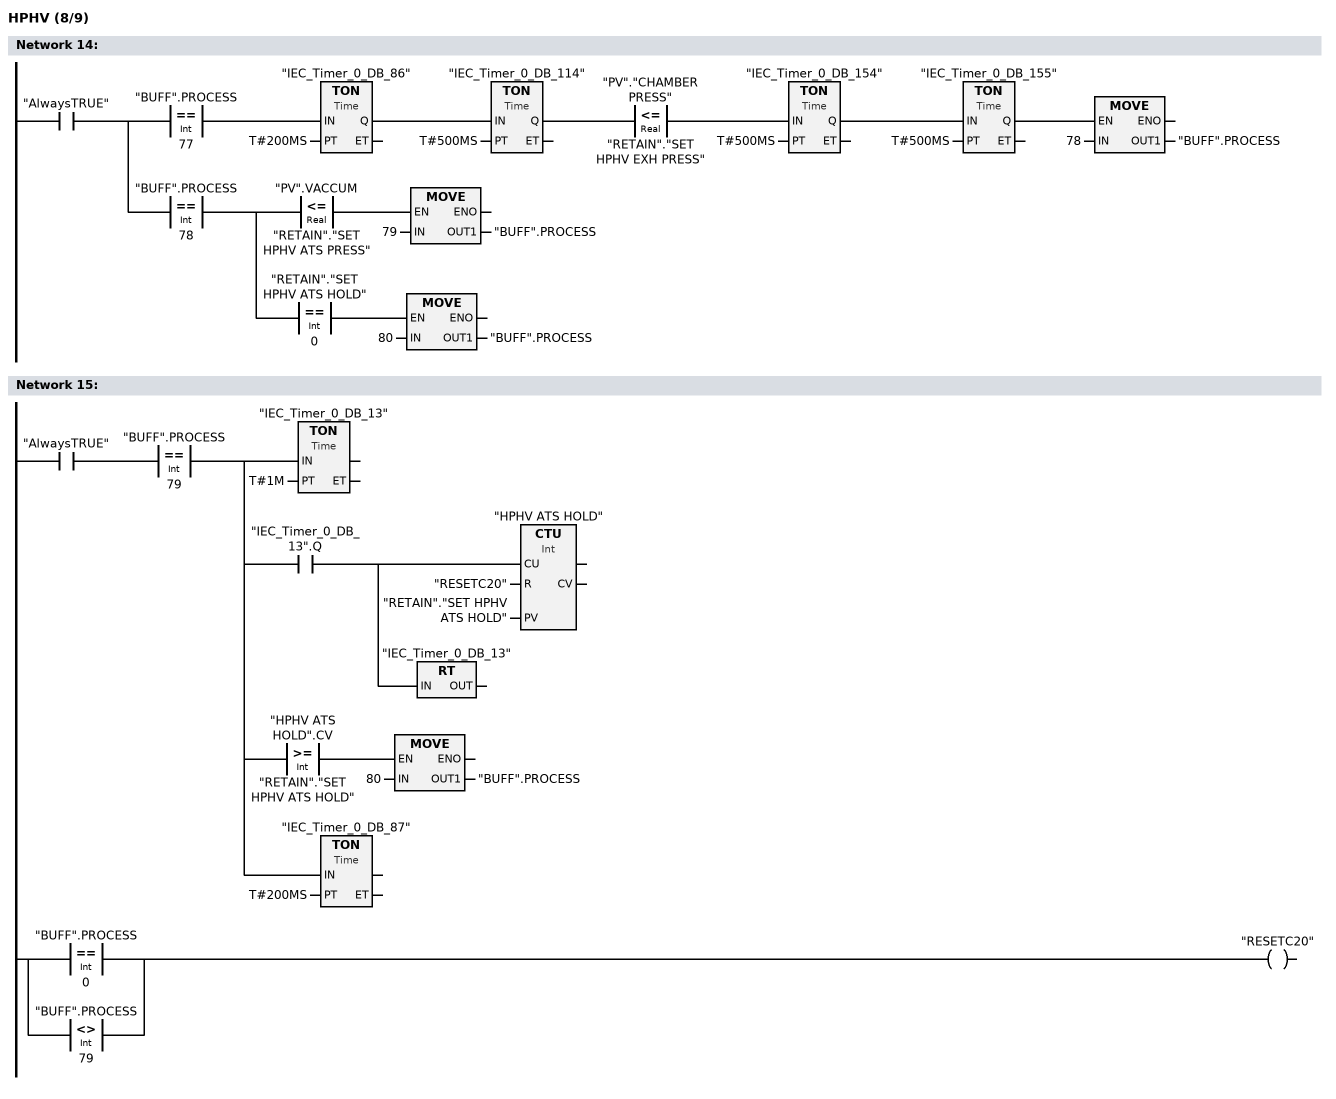
   RUNG wire#powerrail
      Contact( "AlwaysTRUE" )
      wire#w1
      { S7_Templates := "SrcType := Int" } EQ_Contact(in1 := "BUFF".PROCESS, in2 := 77)
      { S7_Templates := "time_type := Time" } "IEC_Timer_0_DB_86".TON(pt := T#200MS, et =>)
      { S7_Templates := "time_type := Time" } "IEC_Timer_0_DB_114".TON(pt := T#500MS, et =>)
      { S7_Templates := "SrcType := Real" } LE_Contact(in1 := "PV"."CHAMBER PRESS", in2 := "RETAIN"."SET HPHV EXH PRESS")
      { S7_Templates := "time_type := Time" } "IEC_Timer_0_DB_154".TON(pt := T#500MS, et =>)
      { S7_Templates := "time_type := Time" } "IEC_Timer_0_DB_155".TON(pt := T#500MS, et =>)
      Move(in := 78, out1 => "BUFF".PROCESS)
   END_RUNG
   RUNG wire#w1
      { S7_Templates := "SrcType := Int" } EQ_Contact(in1 := "BUFF".PROCESS, in2 := 78)
      wire#w2
      { S7_Templates := "SrcType := Real" } LE_Contact(in1 := "PV".VACCUM, in2 := "RETAIN"."SET HPHV ATS PRESS")
      Move(in := 79, out1 => "BUFF".PROCESS)
   END_RUNG
   RUNG wire#w2
      { S7_Templates := "SrcType := Int" } EQ_Contact(in1 := "RETAIN"."SET HPHV ATS HOLD", in2 := 0)
      Move(in := 80, out1 => "BUFF".PROCESS)
   END_RUNG
   // the same network as SCL:
   "IEC_Timer_0_DB_86".TON(IN := "AlwaysTRUE" AND ("BUFF".PROCESS = 77), PT := T#200MS);
   "IEC_Timer_0_DB_114".TON(IN := "IEC_Timer_0_DB_86".Q, PT := T#500MS);
   "IEC_Timer_0_DB_154".TON(IN := "IEC_Timer_0_DB_114".Q AND ("PV"."CHAMBER PRESS" <= "RETAIN"."SET HPHV EXH PRESS"),
                           PT := T#500MS);
   "IEC_Timer_0_DB_155".TON(IN := "IEC_Timer_0_DB_154".Q, PT := T#500MS);
   IF "IEC_Timer_0_DB_155".Q THEN "BUFF".PROCESS := 78; END_IF;
   #_w1 := "AlwaysTRUE" AND ("BUFF".PROCESS = 78);
   IF #_w1 AND ("PV".VACCUM <= "RETAIN"."SET HPHV ATS PRESS") THEN "BUFF".PROCESS := 79; END_IF;
   IF #_w1 AND ("RETAIN"."SET HPHV ATS HOLD" = 0) THEN "BUFF".PROCESS := 80; END_IF;
END_REGION

REGION Network 15
   RUNG wire#powerrail
      Contact( "AlwaysTRUE" )
      { S7_Templates := "SrcType := Int" } EQ_Contact(in1 := "BUFF".PROCESS, in2 := 79)
      wire#w1
      { S7_Templates := "time_type := Time" } "IEC_Timer_0_DB_13".TON(pt := T#1M, et =>)
   END_RUNG
   RUNG wire#w1
      Contact( "IEC_Timer_0_DB_13".Q )
      wire#w2
      { S7_Templates := "value_type := Int" } "HPHV ATS HOLD".CTU(r := "RESETC20", pv := "RETAIN"."SET HPHV ATS HOLD", cv =>)
   END_RUNG
   RUNG wire#w2
      RT_Coil( "IEC_Timer_0_DB_13" )
   END_RUNG
   RUNG wire#w1
      { S7_Templates := "SrcType := Int" } GE_Contact(in1 := "HPHV ATS HOLD".CV, in2 := "RETAIN"."SET HPHV ATS HOLD")
      Move(in := 80, out1 => "BUFF".PROCESS)
   END_RUNG
   RUNG wire#w1
      { S7_Templates := "time_type := Time" } "IEC_Timer_0_DB_87".TON(pt := T#200MS, et =>)
   END_RUNG
   RUNG wire#powerrail
      { S7_Templates := "SrcType := Int" } EQ_Contact(in1 := "BUFF".PROCESS, in2 := 0)
      wire#w3
      Coil( "RESETC20" )
   END_RUNG
   RUNG wire#powerrail
      { S7_Templates := "SrcType := Int" } NE_Contact(in1 := "BUFF".PROCESS, in2 := 79)
   END_RUNG wire#w3
   // the same network as SCL:
   #_w1 := "AlwaysTRUE" AND ("BUFF".PROCESS = 79);
   "IEC_Timer_0_DB_13".TON(IN := #_w1, PT := T#1M);
   #_w2 := #_w1 AND "IEC_Timer_0_DB_13".Q;
   "HPHV ATS HOLD".CTU(CU := #_w2, R := "RESETC20", PV := "RETAIN"."SET HPHV ATS HOLD");
   IF #_w2 THEN RESET_TIMER("IEC_Timer_0_DB_13"); END_IF;
   IF #_w1 AND ("HPHV ATS HOLD".CV >= "RETAIN"."SET HPHV ATS HOLD") THEN "BUFF".PROCESS := 80; END_IF;
   "IEC_Timer_0_DB_87".TON(IN := #_w1, PT := T#200MS);
   "RESETC20" := ("BUFF".PROCESS = 0) OR ("BUFF".PROCESS <> 79);
END_REGION

REGION Network 16
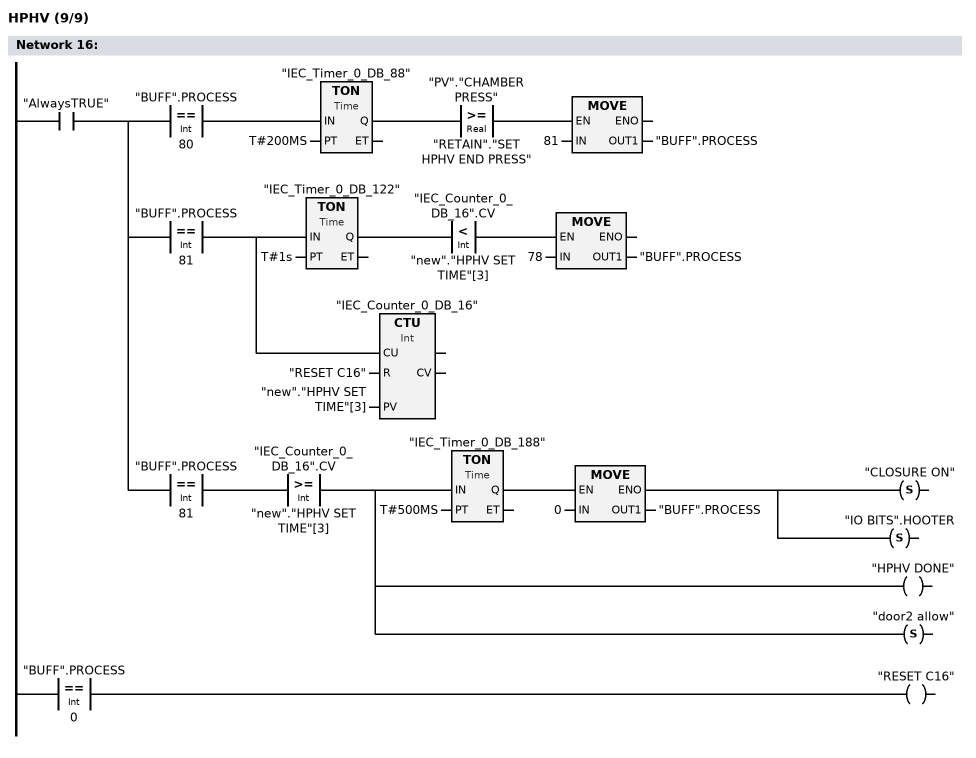
   RUNG wire#powerrail
      Contact( "AlwaysTRUE" )
      wire#w1
      { S7_Templates := "SrcType := Int" } EQ_Contact(in1 := "BUFF".PROCESS, in2 := 80)
      { S7_Templates := "time_type := Time" } "IEC_Timer_0_DB_88".TON(pt := T#200MS, et =>)
      { S7_Templates := "SrcType := Real" } GE_Contact(in1 := "PV"."CHAMBER PRESS", in2 := "RETAIN"."SET HPHV END PRESS")
      Move(in := 81, out1 => "BUFF".PROCESS)
   END_RUNG
   RUNG wire#w1
      { S7_Templates := "SrcType := Int" } EQ_Contact(in1 := "BUFF".PROCESS, in2 := 81)
      wire#w2
      { S7_Templates := "time_type := Time" } "IEC_Timer_0_DB_122".TON(pt := T#1s, et =>)
      { S7_Templates := "SrcType := Int" } LT_Contact(in1 := "IEC_Counter_0_DB_16".CV, in2 := "new"."HPHV SET TIME"[3])
      Move(in := 78, out1 => "BUFF".PROCESS)
   END_RUNG
   RUNG wire#w2
      { S7_Templates := "value_type := Int" } "IEC_Counter_0_DB_16".CTU(r := "RESET C16", pv := "new"."HPHV SET TIME"[3], cv =>)
   END_RUNG
   RUNG wire#w1
      { S7_Templates := "SrcType := Int" } EQ_Contact(in1 := "BUFF".PROCESS, in2 := 81)
      { S7_Templates := "SrcType := Int" } GE_Contact(in1 := "IEC_Counter_0_DB_16".CV, in2 := "new"."HPHV SET TIME"[3])
      wire#w3
      { S7_Templates := "time_type := Time" } "IEC_Timer_0_DB_188".TON(pt := T#500MS, et =>)
      Move(in := 0, out1 => "BUFF".PROCESS)
      wire#w4
      S_Coil( "CLOSURE ON" )
   END_RUNG
   RUNG wire#w4
      S_Coil( "IO BITS".HOOTER )
   END_RUNG
   RUNG wire#w3
      Coil( "HPHV DONE" )
   END_RUNG
   RUNG wire#w3
      S_Coil( "door2 allow" )
   END_RUNG
   RUNG wire#powerrail
      { S7_Templates := "SrcType := Int" } EQ_Contact(in1 := "BUFF".PROCESS, in2 := 0)
      Coil( "RESET C16" )
   END_RUNG
   // the same network as SCL:
   "IEC_Timer_0_DB_88".TON(IN := "AlwaysTRUE" AND ("BUFF".PROCESS = 80), PT := T#200MS);
   IF "IEC_Timer_0_DB_88".Q AND ("PV"."CHAMBER PRESS" >= "RETAIN"."SET HPHV END PRESS") THEN
       "BUFF".PROCESS := 81;
   END_IF;
   #_w1 := "AlwaysTRUE" AND ("BUFF".PROCESS = 81);
   "IEC_Timer_0_DB_122".TON(IN := #_w1, PT := T#1s);
   IF "IEC_Timer_0_DB_122".Q AND ("IEC_Counter_0_DB_16".CV < "new"."HPHV SET TIME"[3]) THEN
       "BUFF".PROCESS := 78;
   END_IF;
   "IEC_Counter_0_DB_16".CTU(CU := #_w1, R := "RESET C16", PV := "new"."HPHV SET TIME"[3]);
   #_w2 := "AlwaysTRUE" AND ("BUFF".PROCESS = 81) AND ("IEC_Counter_0_DB_16".CV >= "new"."HPHV SET TIME"[3]);
   "IEC_Timer_0_DB_188".TON(IN := #_w2, PT := T#500MS);
   IF "IEC_Timer_0_DB_188".Q THEN
       "BUFF".PROCESS := 0;
       "CLOSURE ON" := TRUE;
       "IO BITS".HOOTER := TRUE;
   END_IF;
   "HPHV DONE" := #_w2;
   IF #_w2 THEN "door2 allow" := TRUE; END_IF;
   "RESET C16" := "BUFF".PROCESS = 0;
END_REGION
END_FUNCTION
